TYPE TcaLaserDistanceSenorRef :
STRUCT
	Sensor AT%I* : DINT;	
END_STRUCT
END_TYPE

(* stored: Version 1.1.0.1
   DUT TcaLaserDistanceSenorRef: Id {e32a3552-52d9-4709-8644-fe8858b5ae62} *)
